TYPE ST_AnimationScaling :
STRUCT
END_STRUCT
END_TYPE

(* stored: Version 1.1.0.1, ProductVersion 3.1.4024.10
   DUT ST_AnimationScaling: Id {52811aff-878d-47b5-9418-54d2b8b70faa} *)
